INTERFACE I_Status EXTENDS __SYSTEM.IQueryInterface

PROPERTY CurrentPosition : LREAL
GET
END_GET
END_PROPERTY

PROPERTY CurrentVelocity : LREAL
GET
END_GET
END_PROPERTY

PROPERTY ErrorID : DWORD
GET
END_GET
END_PROPERTY

PROPERTY HasError : BOOL
GET
END_GET
END_PROPERTY

PROPERTY InTargetPosition : BOOL
GET
END_GET
END_PROPERTY

PROPERTY InVelocity : BOOL
GET
END_GET
END_PROPERTY

PROPERTY IsCoupled : bool
GET
END_GET
END_PROPERTY

PROPERTY IsEnabled : bool
GET
END_GET
END_PROPERTY

PROPERTY IsStationary : bool
GET
END_GET
END_PROPERTY

END_INTERFACE

(* stored: Version 1.1.0.1
   Itf I_Status: Id {6057db56-1d8d-4c90-8f15-4379a266ab62}
   Property CurrentPosition: Id {1dd40bc8-3f99-4bad-8e07-083536769e40}
   Get Get: Id {95001c26-a881-4edb-a053-e51c961445d0}
   Property CurrentVelocity: Id {97907787-c05d-4992-abb4-8777b0603fc9}
   Get Get: Id {eb1ce3f9-0501-4350-b473-fbbfd356c617}
   Property ErrorID: Id {b11aa0a0-7098-44ca-82bd-6ca7d22ca21e}
   Get Get: Id {fe8508de-a7df-4935-8954-57d4fdec9685}
   Property HasError: Id {4f9a47cb-8b1f-402d-b2c6-4b52878406bb}
   Get Get: Id {28a41045-34a4-421b-9179-1599bce12a5c}
   Property InTargetPosition: Id {4b369373-838c-4cc4-941b-06225a33951d}
   Get Get: Id {30a64782-fad1-4bf2-a79d-a9c3a2fa8c1e}
   Property InVelocity: Id {89c9aebc-0407-4c60-bfdd-b41bb7aec0a6}
   Get Get: Id {8b2ab8a0-85bf-437a-b651-bf05bdd63e43}
   Property IsCoupled: Id {1482ae7c-1f33-4889-80b5-c5148cec0e70}
   Get Get: Id {f719c339-2597-4343-b354-172be3601a76}
   Property IsEnabled: Id {14fa7212-d544-4f73-a48f-1e9f238c75ce}
   Get Get: Id {601fc560-3c28-4130-bf0b-666aac65d338}
   Property IsStationary: Id {5ca175da-4c6e-4296-8faf-30d6bd78a25a}
   Get Get: Id {50cb22a8-9c64-44df-8969-787a60532850} *)
